       #MyReal	:= 0.0;
       #MyWordsinReal[0]	:= "EPICSToPLC"."Word"[#EPICSToPLCDataBlockOffset + 0];
       #MyWordsinReal[1]	:= "EPICSToPLC"."Word"[#EPICSToPLCDataBlockOffset + 1];
       #"iVolR" := #MyReal;    //EPICSName: iVolR
    Else
       #DEVICE_PARAM_OK := FALSE; //Invalid Hash
    END_IF;
END_FUNCTION_BLOCK
FUNCTION_BLOCK "DEVTYPE_ISRC_LEBT_PS_SOL_STR"
{ S7_Optimized_Access := 'TRUE' }
VERSION : 1.0
   VAR_INPUT
      "CurR-CT" { ExternalAccessible := 'True'; ExternalVisible := 'False'; ExternalWritable := 'False'; } : REAL;   //EPICS Status variable: CurR-CT
      "EnCmdR" { ExternalAccessible := 'True'; ExternalVisible := 'False'; ExternalWritable := 'False'; } : BOOL;   //EPICS Status variable: EnCmdR
      "CurMaxErr" { ExternalAccessible := 'True'; ExternalVisible := 'False'; ExternalWritable := 'False'; } : BOOL;   //EPICS Status variable: CurMaxErr
   EPICSToPLCLength { ExternalAccessible := 'False'; ExternalVisible := 'False'; ExternalWritable := 'False'; } : Int;   // Length of device command register array (in words)
   EPICSToPLCDataBlockOffset { ExternalAccessible := 'False'; ExternalVisible := 'False'; ExternalWritable := 'False'; } : Int;   // Offset in EPICS->PLC comms block where this device data resides (in words)
   EPICSToPLCParametersStart { ExternalAccessible := 'False'; ExternalVisible := 'False'; ExternalWritable := 'False'; } : Int;   // The border offset between the Command and the Parameter area
   PLCToEPICSLength { ExternalAccessible := 'False'; ExternalVisible := 'False'; ExternalWritable := 'False'; } : Int;   // Length of device status register array (in words)
   PLCToEPICSDataBlockOffset { ExternalAccessible := 'False'; ExternalVisible := 'False'; ExternalWritable := 'False'; } : Int;   // Offset in PLC->EPICS comms block where this device data resides (in words)
   END_VAR
   VAR_OUTPUT
      DEVICE_PARAM_OK { ExternalAccessible := 'False'; ExternalVisible := 'False'; ExternalWritable := 'False'; } : Bool;
   END_VAR
   VAR_IN_OUT
   END_VAR
   Var DB_SPECIFIC
      MyWord { ExternalAccessible := 'False'; ExternalVisible := 'False'; ExternalWritable := 'False'; } : Word;
      MyBytesinWord { ExternalAccessible := 'False'; ExternalVisible := 'False'; ExternalWritable := 'False'; } AT MyWord : Array[0..1] of Byte;
      MyBoolsinWord { ExternalAccessible := 'False'; ExternalVisible := 'False'; ExternalWritable := 'False'; } AT MyWord : Array[0..15] of Bool;
      MyDInt { ExternalAccessible := 'False'; ExternalVisible := 'False'; ExternalWritable := 'False'; } : DInt;
      MyWordsinDint { ExternalAccessible := 'False'; ExternalVisible := 'False'; ExternalWritable := 'False'; } AT MyDInt : Array[0..1] of Word;
      MyReal { ExternalAccessible := 'False'; ExternalVisible := 'False'; ExternalWritable := 'False'; } : Real;
      MyWordsinReal { ExternalAccessible := 'False'; ExternalVisible := 'False'; ExternalWritable := 'False'; } AT MyReal : Array[0..1] of Word;
      MyInt { ExternalAccessible := 'False'; ExternalVisible := 'False'; ExternalWritable := 'False'; } : Int;
      MyWordinInt { ExternalAccessible := 'False'; ExternalVisible := 'False'; ExternalWritable := 'False'; } AT MyInt : Word;
      MyDWord { ExternalAccessible := 'False'; ExternalVisible := 'False'; ExternalWritable := 'False'; } : DWord;
      MyWordsinDWord { ExternalAccessible := 'False'; ExternalVisible := 'False'; ExternalWritable := 'False'; } AT MyDWord : Array[0..1] of Word;
      MyTime { ExternalAccessible := 'False'; ExternalVisible := 'False'; ExternalWritable := 'False'; } : Time;
      MyWordsinTime { ExternalAccessible := 'False'; ExternalVisible := 'False'; ExternalWritable := 'False'; } AT MyTime : Array[0..1] of Word;
      MyString { ExternalAccessible := 'False'; ExternalVisible := 'False'; ExternalWritable := 'False'; } : String[40];
      MyWordsinString { ExternalAccessible := 'False'; ExternalVisible := 'False'; ExternalWritable := 'False'; } AT MyString : Array[0..20] of Word;
   END_VAR
   VAR_TEMP
      HashModbus : DInt;
      HashIFA : DInt;
      HashTIAMap : DInt;
      i : Int;
   END_VAR
    //Author: Miklos Boros (miklos.boros@esss.se), Copyrigth 2017-2019 by European Spallation Source, Lund
    //This block was generated by PLCFactory, please don't change it MANUALLY!
    //Input File Name: ISrc-010_Ctrl-PLC-01-template-IFA-20191106135317.ifa
    //Generated: 20191106135317
    //According to HASH: 1347332123
    //Device type: ISRC_LEBT_PS_SOL_STR
    //Description: This function does the variable mapping for a device. All device-variable will be linked to an interface variable defined in this block.

    //********************************************
    //****************HASH check******************
    //********************************************


    #MyWordsinDint[0] := "EPICSToPLC"."Word"[0];
    #MyWordsinDint[1] := "EPICSToPLC"."Word"[1];
    #HashModbus := #MyDInt; //Hash from EPICS/ModbusTCP

    #HashIFA := 1347332123; //Hash from Interface Factory as a constant

    #MyWordsinDint[0] := "PLCToEPICS"."Word"[0];
    #MyWordsinDint[1] := "PLCToEPICS"."Word"[1];
    #HashTIAMap := #MyDInt; //Hash from PLCFactory TIA Map


    IF ((#HashIFA = #HashModbus) AND (#HashModbus = #HashTIAMap)) THEN //Check CRCs
        #DEVICE_PARAM_OK := TRUE;
       //###########################  LEBT Solenoids and Steerers PowerSupply  ##############################
       //###########################
       //STATUS BLOCK
       //###########################

    //********************************************
    //*************STATUS VARIABLES***************
    //********************************************


       #MyReal := #"CurR-CT";    //EPICSName: CurR-CT
       "PLCToEPICS"."Word"[#PLCToEPICSDataBlockOffset + 0] := #MyWordsinReal[0];
       "PLCToEPICS"."Word"[#PLCToEPICSDataBlockOffset + 1] := #MyWordsinReal[1];

       #MyWord := W#0;
       #MyBoolsinWord[8] := #"EnCmdR";    //EPICSName: EnCmdR
       #MyBoolsinWord[9] := #"CurMaxErr";    //EPICSName: CurMaxErr
       "PLCToEPICS"."Word"[#PLCToEPICSDataBlockOffset + 2] := #MyWord;
    Else
       #DEVICE_PARAM_OK := FALSE; //Invalid Hash
    END_IF;
END_FUNCTION_BLOCK
FUNCTION_BLOCK "DEVTYPE_ISRC_LEBT_PlasCh"
{ S7_Optimized_Access := 'TRUE' }
VERSION : 1.0
   VAR_INPUT
      "WtrFlowOK" { ExternalAccessible := 'True'; ExternalVisible := 'False'; ExternalWritable := 'False'; } : BOOL;   //EPICS Status variable: WtrFlowOK
   EPICSToPLCLength { ExternalAccessible := 'False'; ExternalVisible := 'False'; ExternalWritable := 'False'; } : Int;   // Length of device command register array (in words)
   EPICSToPLCDataBlockOffset { ExternalAccessible := 'False'; ExternalVisible := 'False'; ExternalWritable := 'False'; } : Int;   // Offset in EPICS->PLC comms block where this device data resides (in words)
   EPICSToPLCParametersStart { ExternalAccessible := 'False'; ExternalVisible := 'False'; ExternalWritable := 'False'; } : Int;   // The border offset between the Command and the Parameter area
   PLCToEPICSLength { ExternalAccessible := 'False'; ExternalVisible := 'False'; ExternalWritable := 'False'; } : Int;   // Length of device status register array (in words)
   PLCToEPICSDataBlockOffset { ExternalAccessible := 'False'; ExternalVisible := 'False'; ExternalWritable := 'False'; } : Int;   // Offset in PLC->EPICS comms block where this device data resides (in words)
   END_VAR
   VAR_OUTPUT
      DEVICE_PARAM_OK { ExternalAccessible := 'False'; ExternalVisible := 'False'; ExternalWritable := 'False'; } : Bool;
   END_VAR
   VAR_IN_OUT
   END_VAR
   Var DB_SPECIFIC
      MyWord { ExternalAccessible := 'False'; ExternalVisible := 'False'; ExternalWritable := 'False'; } : Word;
      MyBytesinWord { ExternalAccessible := 'False'; ExternalVisible := 'False'; ExternalWritable := 'False'; } AT MyWord : Array[0..1] of Byte;
      MyBoolsinWord { ExternalAccessible := 'False'; ExternalVisible := 'False'; ExternalWritable := 'False'; } AT MyWord : Array[0..15] of Bool;
      MyDInt { ExternalAccessible := 'False'; ExternalVisible := 'False'; ExternalWritable := 'False'; } : DInt;
      MyWordsinDint { ExternalAccessible := 'False'; ExternalVisible := 'False'; ExternalWritable := 'False'; } AT MyDInt : Array[0..1] of Word;
      MyReal { ExternalAccessible := 'False'; ExternalVisible := 'False'; ExternalWritable := 'False'; } : Real;
      MyWordsinReal { ExternalAccessible := 'False'; ExternalVisible := 'False'; ExternalWritable := 'False'; } AT MyReal : Array[0..1] of Word;
      MyInt { ExternalAccessible := 'False'; ExternalVisible := 'False'; ExternalWritable := 'False'; } : Int;
      MyWordinInt { ExternalAccessible := 'False'; ExternalVisible := 'False'; ExternalWritable := 'False'; } AT MyInt : Word;
      MyDWord { ExternalAccessible := 'False'; ExternalVisible := 'False'; ExternalWritable := 'False'; } : DWord;
      MyWordsinDWord { ExternalAccessible := 'False'; ExternalVisible := 'False'; ExternalWritable := 'False'; } AT MyDWord : Array[0..1] of Word;
      MyTime { ExternalAccessible := 'False'; ExternalVisible := 'False'; ExternalWritable := 'False'; } : Time;
      MyWordsinTime { ExternalAccessible := 'False'; ExternalVisible := 'False'; ExternalWritable := 'False'; } AT MyTime : Array[0..1] of Word;
      MyString { ExternalAccessible := 'False'; ExternalVisible := 'False'; ExternalWritable := 'False'; } : String[40];
      MyWordsinString { ExternalAccessible := 'False'; ExternalVisible := 'False'; ExternalWritable := 'False'; } AT MyString : Array[0..20] of Word;
   END_VAR
   VAR_TEMP
      HashModbus : DInt;
      HashIFA : DInt;
      HashTIAMap : DInt;
      i : Int;
   END_VAR
    //Author: Miklos Boros (miklos.boros@esss.se), Copyrigth 2017-2019 by European Spallation Source, Lund
    //This block was generated by PLCFactory, please don't change it MANUALLY!
    //Input File Name: ISrc-010_Ctrl-PLC-01-template-IFA-20191106135317.ifa
    //Generated: 20191106135317
    //According to HASH: 1347332123
    //Device type: ISRC_LEBT_PlasCh
    //Description: This function does the variable mapping for a device. All device-variable will be linked to an interface variable defined in this block.

    //********************************************
    //****************HASH check******************
    //********************************************


    #MyWordsinDint[0] := "EPICSToPLC"."Word"[0];
    #MyWordsinDint[1] := "EPICSToPLC"."Word"[1];
    #HashModbus := #MyDInt; //Hash from EPICS/ModbusTCP

    #HashIFA := 1347332123; //Hash from Interface Factory as a constant

    #MyWordsinDint[0] := "PLCToEPICS"."Word"[0];
    #MyWordsinDint[1] := "PLCToEPICS"."Word"[1];
    #HashTIAMap := #MyDInt; //Hash from PLCFactory TIA Map


    IF ((#HashIFA = #HashModbus) AND (#HashModbus = #HashTIAMap)) THEN //Check CRCs
        #DEVICE_PARAM_OK := TRUE;
       //###########################  ISRC Plasma Chamber  ##############################
       //###########################
       //STATUS BLOCK
       //###########################

    //********************************************
    //*************STATUS VARIABLES***************
    //********************************************


       #MyWord := W#0;
       #MyBoolsinWord[8] := #"WtrFlowOK";    //EPICSName: WtrFlowOK
       "PLCToEPICS"."Word"[#PLCToEPICSDataBlockOffset + 0] := #MyWord;
    Else
       #DEVICE_PARAM_OK := FALSE; //Invalid Hash
    END_IF;
END_FUNCTION_BLOCK
FUNCTION_BLOCK "DEVTYPE_ISRC_LEBT_REP"
{ S7_Optimized_Access := 'TRUE' }
VERSION : 1.0
   VAR_INPUT
      "WtrFlowOK" { ExternalAccessible := 'True'; ExternalVisible := 'False'; ExternalWritable := 'False'; } : BOOL;   //EPICS Status variable: WtrFlowOK
   EPICSToPLCLength { ExternalAccessible := 'False'; ExternalVisible := 'False'; ExternalWritable := 'False'; } : Int;   // Length of device command register array (in words)
   EPICSToPLCDataBlockOffset { ExternalAccessible := 'False'; ExternalVisible := 'False'; ExternalWritable := 'False'; } : Int;   // Offset in EPICS->PLC comms block where this device data resides (in words)
   EPICSToPLCParametersStart { ExternalAccessible := 'False'; ExternalVisible := 'False'; ExternalWritable := 'False'; } : Int;   // The border offset between the Command and the Parameter area
   PLCToEPICSLength { ExternalAccessible := 'False'; ExternalVisible := 'False'; ExternalWritable := 'False'; } : Int;   // Length of device status register array (in words)
   PLCToEPICSDataBlockOffset { ExternalAccessible := 'False'; ExternalVisible := 'False'; ExternalWritable := 'False'; } : Int;   // Offset in PLC->EPICS comms block where this device data resides (in words)
   END_VAR
   VAR_OUTPUT
      DEVICE_PARAM_OK { ExternalAccessible := 'False'; ExternalVisible := 'False'; ExternalWritable := 'False'; } : Bool;
   END_VAR
   VAR_IN_OUT
   END_VAR
   Var DB_SPECIFIC
      MyWord { ExternalAccessible := 'False'; ExternalVisible := 'False'; ExternalWritable := 'False'; } : Word;
      MyBytesinWord { ExternalAccessible := 'False'; ExternalVisible := 'False'; ExternalWritable := 'False'; } AT MyWord : Array[0..1] of Byte;
      MyBoolsinWord { ExternalAccessible := 'False'; ExternalVisible := 'False'; ExternalWritable := 'False'; } AT MyWord : Array[0..15] of Bool;
      MyDInt { ExternalAccessible := 'False'; ExternalVisible := 'False'; ExternalWritable := 'False'; } : DInt;
      MyWordsinDint { ExternalAccessible := 'False'; ExternalVisible := 'False'; ExternalWritable := 'False'; } AT MyDInt : Array[0..1] of Word;
      MyReal { ExternalAccessible := 'False'; ExternalVisible := 'False'; ExternalWritable := 'False'; } : Real;
      MyWordsinReal { ExternalAccessible := 'False'; ExternalVisible := 'False'; ExternalWritable := 'False'; } AT MyReal : Array[0..1] of Word;
      MyInt { ExternalAccessible := 'False'; ExternalVisible := 'False'; ExternalWritable := 'False'; } : Int;
      MyWordinInt { ExternalAccessible := 'False'; ExternalVisible := 'False'; ExternalWritable := 'False'; } AT MyInt : Word;
      MyDWord { ExternalAccessible := 'False'; ExternalVisible := 'False'; ExternalWritable := 'False'; } : DWord;
      MyWordsinDWord { ExternalAccessible := 'False'; ExternalVisible := 'False'; ExternalWritable := 'False'; } AT MyDWord : Array[0..1] of Word;
      MyTime { ExternalAccessible := 'False'; ExternalVisible := 'False'; ExternalWritable := 'False'; } : Time;
      MyWordsinTime { ExternalAccessible := 'False'; ExternalVisible := 'False'; ExternalWritable := 'False'; } AT MyTime : Array[0..1] of Word;
      MyString { ExternalAccessible := 'False'; ExternalVisible := 'False'; ExternalWritable := 'False'; } : String[40];
      MyWordsinString { ExternalAccessible := 'False'; ExternalVisible := 'False'; ExternalWritable := 'False'; } AT MyString : Array[0..20] of Word;
   END_VAR
   VAR_TEMP
      HashModbus : DInt;
      HashIFA : DInt;
      HashTIAMap : DInt;
      i : Int;
   END_VAR
    //Author: Miklos Boros (miklos.boros@esss.se), Copyrigth 2017-2019 by European Spallation Source, Lund
    //This block was generated by PLCFactory, please don't change it MANUALLY!
    //Input File Name: ISrc-010_Ctrl-PLC-01-template-IFA-20191106135317.ifa
    //Generated: 20191106135317
    //According to HASH: 1347332123
    //Device type: ISRC_LEBT_REP
    //Description: This function does the variable mapping for a device. All device-variable will be linked to an interface variable defined in this block.

    //********************************************
    //****************HASH check******************
    //********************************************


    #MyWordsinDint[0] := "EPICSToPLC"."Word"[0];
    #MyWordsinDint[1] := "EPICSToPLC"."Word"[1];
    #HashModbus := #MyDInt; //Hash from EPICS/ModbusTCP

    #HashIFA := 1347332123; //Hash from Interface Factory as a constant

    #MyWordsinDint[0] := "PLCToEPICS"."Word"[0];
    #MyWordsinDint[1] := "PLCToEPICS"."Word"[1];
    #HashTIAMap := #MyDInt; //Hash from PLCFactory TIA Map


    IF ((#HashIFA = #HashModbus) AND (#HashModbus = #HashTIAMap)) THEN //Check CRCs
        #DEVICE_PARAM_OK := TRUE;
       //###########################  ISrc and LEBT Repeller  ##############################
       //###########################
       //STATUS BLOCK
       //###########################

    //********************************************
    //*************STATUS VARIABLES***************
    //********************************************


       #MyWord := W#0;
       #MyBoolsinWord[8] := #"WtrFlowOK";    //EPICSName: WtrFlowOK
       "PLCToEPICS"."Word"[#PLCToEPICSDataBlockOffset + 0] := #MyWord;
    Else
       #DEVICE_PARAM_OK := FALSE; //Invalid Hash
    END_IF;
END_FUNCTION_BLOCK
FUNCTION_BLOCK "DEVTYPE_ISRC_LEBT_STR"
{ S7_Optimized_Access := 'TRUE' }
VERSION : 1.0
   VAR_INPUT
      "PolR" { ExternalAccessible := 'True'; ExternalVisible := 'False'; ExternalWritable := 'False'; } : BOOL;   //EPICS Status variable: PolR
   EPICSToPLCLength { ExternalAccessible := 'False'; ExternalVisible := 'False'; ExternalWritable := 'False'; } : Int;   // Length of device command register array (in words)
   EPICSToPLCDataBlockOffset { ExternalAccessible := 'False'; ExternalVisible := 'False'; ExternalWritable := 'False'; } : Int;   // Offset in EPICS->PLC comms block where this device data resides (in words)
   EPICSToPLCParametersStart { ExternalAccessible := 'False'; ExternalVisible := 'False'; ExternalWritable := 'False'; } : Int;   // The border offset between the Command and the Parameter area
   PLCToEPICSLength { ExternalAccessible := 'False'; ExternalVisible := 'False'; ExternalWritable := 'False'; } : Int;   // Length of device status register array (in words)
   PLCToEPICSDataBlockOffset { ExternalAccessible := 'False'; ExternalVisible := 'False'; ExternalWritable := 'False'; } : Int;   // Offset in PLC->EPICS comms block where this device data resides (in words)
   END_VAR
   VAR_OUTPUT
      "PolPosCmd" { ExternalAccessible := 'True'; ExternalVisible := 'False'; ExternalWritable := 'False'; } : BOOL;   //EPICS Command variable: PolPosCmd
      "PolNegCmd" { ExternalAccessible := 'True'; ExternalVisible := 'False'; ExternalWritable := 'False'; } : BOOL;   //EPICS Command variable: PolNegCmd
      DEVICE_PARAM_OK { ExternalAccessible := 'False'; ExternalVisible := 'False'; ExternalWritable := 'False'; } : Bool;
   END_VAR
   VAR_IN_OUT
   END_VAR
   Var DB_SPECIFIC
      MyWord { ExternalAccessible := 'False'; ExternalVisible := 'False'; ExternalWritable := 'False'; } : Word;
      MyBytesinWord { ExternalAccessible := 'False'; ExternalVisible := 'False'; ExternalWritable := 'False'; } AT MyWord : Array[0..1] of Byte;
      MyBoolsinWord { ExternalAccessible := 'False'; ExternalVisible := 'False'; ExternalWritable := 'False'; } AT MyWord : Array[0..15] of Bool;
      MyDInt { ExternalAccessible := 'False'; ExternalVisible := 'False'; ExternalWritable := 'False'; } : DInt;
      MyWordsinDint { ExternalAccessible := 'False'; ExternalVisible := 'False'; ExternalWritable := 'False'; } AT MyDInt : Array[0..1] of Word;
      MyReal { ExternalAccessible := 'False'; ExternalVisible := 'False'; ExternalWritable := 'False'; } : Real;
      MyWordsinReal { ExternalAccessible := 'False'; ExternalVisible := 'False'; ExternalWritable := 'False'; } AT MyReal : Array[0..1] of Word;
      MyInt { ExternalAccessible := 'False'; ExternalVisible := 'False'; ExternalWritable := 'False'; } : Int;
      MyWordinInt { ExternalAccessible := 'False'; ExternalVisible := 'False'; ExternalWritable := 'False'; } AT MyInt : Word;
      MyDWord { ExternalAccessible := 'False'; ExternalVisible := 'False'; ExternalWritable := 'False'; } : DWord;
      MyWordsinDWord { ExternalAccessible := 'False'; ExternalVisible := 'False'; ExternalWritable := 'False'; } AT MyDWord : Array[0..1] of Word;
      MyTime { ExternalAccessible := 'False'; ExternalVisible := 'False'; ExternalWritable := 'False'; } : Time;
      MyWordsinTime { ExternalAccessible := 'False'; ExternalVisible := 'False'; ExternalWritable := 'False'; } AT MyTime : Array[0..1] of Word;
      MyString { ExternalAccessible := 'False'; ExternalVisible := 'False'; ExternalWritable := 'False'; } : String[40];
      MyWordsinString { ExternalAccessible := 'False'; ExternalVisible := 'False'; ExternalWritable := 'False'; } AT MyString : Array[0..20] of Word;
   END_VAR
   VAR_TEMP
      HashModbus : DInt;
      HashIFA : DInt;
      HashTIAMap : DInt;
      i : Int;
   END_VAR
    //Author: Miklos Boros (miklos.boros@esss.se), Copyrigth 2017-2019 by European Spallation Source, Lund
    //This block was generated by PLCFactory, please don't change it MANUALLY!
    //Input File Name: ISrc-010_Ctrl-PLC-01-template-IFA-20191106135317.ifa
    //Generated: 20191106135317
    //According to HASH: 1347332123
    //Device type: ISRC_LEBT_STR
    //Description: This function does the variable mapping for a device. All device-variable will be linked to an interface variable defined in this block.

    //********************************************
    //****************HASH check******************
    //********************************************


    #MyWordsinDint[0] := "EPICSToPLC"."Word"[0];
    #MyWordsinDint[1] := "EPICSToPLC"."Word"[1];
    #HashModbus := #MyDInt; //Hash from EPICS/ModbusTCP

    #HashIFA := 1347332123; //Hash from Interface Factory as a constant

    #MyWordsinDint[0] := "PLCToEPICS"."Word"[0];
    #MyWordsinDint[1] := "PLCToEPICS"."Word"[1];
    #HashTIAMap := #MyDInt; //Hash from PLCFactory TIA Map


    IF ((#HashIFA = #HashModbus) AND (#HashModbus = #HashTIAMap)) THEN //Check CRCs
        #DEVICE_PARAM_OK := TRUE;
       //#############################  LEBT Steerer  ##############################
       //###########################
       //STATUS BLOCK
       //###########################

    //********************************************
    //*************STATUS VARIABLES***************
    //********************************************


       #MyWord := W#0;
       #MyBoolsinWord[8] := #"PolR";    //EPICSName: PolR
       "PLCToEPICS"."Word"[#PLCToEPICSDataBlockOffset + 0] := #MyWord;

    //********************************************
    //*************COMMAND VARIABLES**************
    //********************************************


       #MyWord := "EPICSToPLC"."Word"[#EPICSToPLCDataBlockOffset + 0];
       IF (NOT "Utilities".TestInProgress) THEN
       	"EPICSToPLC"."Word"[#EPICSToPLCDataBlockOffset + 0] := 0;
       END_IF;
       #"PolPosCmd" := #MyBoolsinWord[8];    //EPICSName: PolPosCmd
       #"PolNegCmd" := #MyBoolsinWord[9];    //EPICSName: PolNegCmd
    Else
       #DEVICE_PARAM_OK := FALSE; //Invalid Hash
    END_IF;
END_FUNCTION_BLOCK
FUNCTION_BLOCK "DEVTYPE_ISRC_LEBT_VAC_VVA"
{ S7_Optimized_Access := 'TRUE' }
VERSION : 1.0
   VAR_INPUT
      "OpenR" { ExternalAccessible := 'True'; ExternalVisible := 'False'; ExternalWritable := 'False'; } : BOOL;   //EPICS Status variable: OpenR
      "OpenCmdRB" { ExternalAccessible := 'True'; ExternalVisible := 'False'; ExternalWritable := 'False'; } : BOOL;   //EPICS Status variable: OpenCmdRB
   EPICSToPLCLength { ExternalAccessible := 'False'; ExternalVisible := 'False'; ExternalWritable := 'False'; } : Int;   // Length of device command register array (in words)
   EPICSToPLCDataBlockOffset { ExternalAccessible := 'False'; ExternalVisible := 'False'; ExternalWritable := 'False'; } : Int;   // Offset in EPICS->PLC comms block where this device data resides (in words)
   EPICSToPLCParametersStart { ExternalAccessible := 'False'; ExternalVisible := 'False'; ExternalWritable := 'False'; } : Int;   // The border offset between the Command and the Parameter area
   PLCToEPICSLength { ExternalAccessible := 'False'; ExternalVisible := 'False'; ExternalWritable := 'False'; } : Int;   // Length of device status register array (in words)
   PLCToEPICSDataBlockOffset { ExternalAccessible := 'False'; ExternalVisible := 'False'; ExternalWritable := 'False'; } : Int;   // Offset in PLC->EPICS comms block where this device data resides (in words)
   END_VAR
   VAR_OUTPUT
      "OpenCmd" { ExternalAccessible := 'True'; ExternalVisible := 'False'; ExternalWritable := 'False'; } : BOOL;   //EPICS Command variable: OpenCmd
      "CloseCmd" { ExternalAccessible := 'True'; ExternalVisible := 'False'; ExternalWritable := 'False'; } : BOOL;   //EPICS Command variable: CloseCmd
      DEVICE_PARAM_OK { ExternalAccessible := 'False'; ExternalVisible := 'False'; ExternalWritable := 'False'; } : Bool;
   END_VAR
   VAR_IN_OUT
   END_VAR
   Var DB_SPECIFIC
      MyWord { ExternalAccessible := 'False'; ExternalVisible := 'False'; ExternalWritable := 'False'; } : Word;
      MyBytesinWord { ExternalAccessible := 'False'; ExternalVisible := 'False'; ExternalWritable := 'False'; } AT MyWord : Array[0..1] of Byte;
      MyBoolsinWord { ExternalAccessible := 'False'; ExternalVisible := 'False'; ExternalWritable := 'False'; } AT MyWord : Array[0..15] of Bool;
      MyDInt { ExternalAccessible := 'False'; ExternalVisible := 'False'; ExternalWritable := 'False'; } : DInt;
      MyWordsinDint { ExternalAccessible := 'False'; ExternalVisible := 'False'; ExternalWritable := 'False'; } AT MyDInt : Array[0..1] of Word;
      MyReal { ExternalAccessible := 'False'; ExternalVisible := 'False'; ExternalWritable := 'False'; } : Real;
      MyWordsinReal { ExternalAccessible := 'False'; ExternalVisible := 'False'; ExternalWritable := 'False'; } AT MyReal : Array[0..1] of Word;
      MyInt { ExternalAccessible := 'False'; ExternalVisible := 'False'; ExternalWritable := 'False'; } : Int;
      MyWordinInt { ExternalAccessible := 'False'; ExternalVisible := 'False'; ExternalWritable := 'False'; } AT MyInt : Word;
      MyDWord { ExternalAccessible := 'False'; ExternalVisible := 'False'; ExternalWritable := 'False'; } : DWord;
      MyWordsinDWord { ExternalAccessible := 'False'; ExternalVisible := 'False'; ExternalWritable := 'False'; } AT MyDWord : Array[0..1] of Word;
      MyTime { ExternalAccessible := 'False'; ExternalVisible := 'False'; ExternalWritable := 'False'; } : Time;
      MyWordsinTime { ExternalAccessible := 'False'; ExternalVisible := 'False'; ExternalWritable := 'False'; } AT MyTime : Array[0..1] of Word;
      MyString { ExternalAccessible := 'False'; ExternalVisible := 'False'; ExternalWritable := 'False'; } : String[40];
      MyWordsinString { ExternalAccessible := 'False'; ExternalVisible := 'False'; ExternalWritable := 'False'; } AT MyString : Array[0..20] of Word;
   END_VAR
   VAR_TEMP
      HashModbus : DInt;
      HashIFA : DInt;
      HashTIAMap : DInt;
      i : Int;
   END_VAR
    //Author: Miklos Boros (miklos.boros@esss.se), Copyrigth 2017-2019 by European Spallation Source, Lund
    //This block was generated by PLCFactory, please don't change it MANUALLY!
    //Input File Name: ISrc-010_Ctrl-PLC-01-template-IFA-20191106135317.ifa
    //Generated: 20191106135317
    //According to HASH: 1347332123
    //Device type: ISRC_LEBT_VAC_VVA
    //Description: This function does the variable mapping for a device. All device-variable will be linked to an interface variable defined in this block.

    //********************************************
    //****************HASH check******************
    //********************************************


    #MyWordsinDint[0] := "EPICSToPLC"."Word"[0];
    #MyWordsinDint[1] := "EPICSToPLC"."Word"[1];
    #HashModbus := #MyDInt; //Hash from EPICS/ModbusTCP

    #HashIFA := 1347332123; //Hash from Interface Factory as a constant

    #MyWordsinDint[0] := "PLCToEPICS"."Word"[0];
    #MyWordsinDint[1] := "PLCToEPICS"."Word"[1];
    #HashTIAMap := #MyDInt; //Hash from PLCFactory TIA Map


    IF ((#HashIFA = #HashModbus) AND (#HashModbus = #HashTIAMap)) THEN //Check CRCs
        #DEVICE_PARAM_OK := TRUE;
       //###########################  ISRC_LEBT H2 valve in HV platform  ##############################
       //###########################
       //STATUS BLOCK
       //###########################

    //********************************************
    //*************STATUS VARIABLES***************
    //********************************************


       #MyWord := W#0;
       #MyBoolsinWord[8] := #"OpenR";    //EPICSName: OpenR
       #MyBoolsinWord[9] := #"OpenCmdRB";    //EPICSName: OpenCmdRB
       "PLCToEPICS"."Word"[#PLCToEPICSDataBlockOffset + 0] := #MyWord;

    //********************************************
    //*************COMMAND VARIABLES**************
    //********************************************


       #MyWord := "EPICSToPLC"."Word"[#EPICSToPLCDataBlockOffset + 0];
       IF (NOT "Utilities".TestInProgress) THEN
       	"EPICSToPLC"."Word"[#EPICSToPLCDataBlockOffset + 0] := 0;
       END_IF;
       #"OpenCmd" := #MyBoolsinWord[8];    //EPICSName: OpenCmd
       #"CloseCmd" := #MyBoolsinWord[9];    //EPICSName: CloseCmd
    Else
       #DEVICE_PARAM_OK := FALSE; //Invalid Hash
    END_IF;
END_FUNCTION_BLOCK
FUNCTION_BLOCK "DEVTYPE_ISRC_LEBT_WTRC_PRES"
{ S7_Optimized_Access := 'TRUE' }
VERSION : 1.0
   VAR_INPUT
      "PresR" { ExternalAccessible := 'True'; ExternalVisible := 'False'; ExternalWritable := 'False'; } : REAL;   //EPICS Status variable: PresR
   EPICSToPLCLength { ExternalAccessible := 'False'; ExternalVisible := 'False'; ExternalWritable := 'False'; } : Int;   // Length of device command register array (in words)
   EPICSToPLCDataBlockOffset { ExternalAccessible := 'False'; ExternalVisible := 'False'; ExternalWritable := 'False'; } : Int;   // Offset in EPICS->PLC comms block where this device data resides (in words)
   EPICSToPLCParametersStart { ExternalAccessible := 'False'; ExternalVisible := 'False'; ExternalWritable := 'False'; } : Int;   // The border offset between the Command and the Parameter area
   PLCToEPICSLength { ExternalAccessible := 'False'; ExternalVisible := 'False'; ExternalWritable := 'False'; } : Int;   // Length of device status register array (in words)
   PLCToEPICSDataBlockOffset { ExternalAccessible := 'False'; ExternalVisible := 'False'; ExternalWritable := 'False'; } : Int;   // Offset in PLC->EPICS comms block where this device data resides (in words)
   END_VAR
   VAR_OUTPUT
      DEVICE_PARAM_OK { ExternalAccessible := 'False'; ExternalVisible := 'False'; ExternalWritable := 'False'; } : Bool;
   END_VAR
   VAR_IN_OUT
   END_VAR
   Var DB_SPECIFIC
      MyWord { ExternalAccessible := 'False'; ExternalVisible := 'False'; ExternalWritable := 'False'; } : Word;
      MyBytesinWord { ExternalAccessible := 'False'; ExternalVisible := 'False'; ExternalWritable := 'False'; } AT MyWord : Array[0..1] of Byte;
      MyBoolsinWord { ExternalAccessible := 'False'; ExternalVisible := 'False'; ExternalWritable := 'False'; } AT MyWord : Array[0..15] of Bool;
      MyDInt { ExternalAccessible := 'False'; ExternalVisible := 'False'; ExternalWritable := 'False'; } : DInt;
      MyWordsinDint { ExternalAccessible := 'False'; ExternalVisible := 'False'; ExternalWritable := 'False'; } AT MyDInt : Array[0..1] of Word;
      MyReal { ExternalAccessible := 'False'; ExternalVisible := 'False'; ExternalWritable := 'False'; } : Real;
      MyWordsinReal { ExternalAccessible := 'False'; ExternalVisible := 'False'; ExternalWritable := 'False'; } AT MyReal : Array[0..1] of Word;
      MyInt { ExternalAccessible := 'False'; ExternalVisible := 'False'; ExternalWritable := 'False'; } : Int;
      MyWordinInt { ExternalAccessible := 'False'; ExternalVisible := 'False'; ExternalWritable := 'False'; } AT MyInt : Word;
      MyDWord { ExternalAccessible := 'False'; ExternalVisible := 'False'; ExternalWritable := 'False'; } : DWord;
      MyWordsinDWord { ExternalAccessible := 'False'; ExternalVisible := 'False'; ExternalWritable := 'False'; } AT MyDWord : Array[0..1] of Word;
      MyTime { ExternalAccessible := 'False'; ExternalVisible := 'False'; ExternalWritable := 'False'; } : Time;
      MyWordsinTime { ExternalAccessible := 'False'; ExternalVisible := 'False'; ExternalWritable := 'False'; } AT MyTime : Array[0..1] of Word;
      MyString { ExternalAccessible := 'False'; ExternalVisible := 'False'; ExternalWritable := 'False'; } : String[40];
      MyWordsinString { ExternalAccessible := 'False'; ExternalVisible := 'False'; ExternalWritable := 'False'; } AT MyString : Array[0..20] of Word;
   END_VAR
   VAR_TEMP
      HashModbus : DInt;
      HashIFA : DInt;
      HashTIAMap : DInt;
      i : Int;
   END_VAR
    //Author: Miklos Boros (miklos.boros@esss.se), Copyrigth 2017-2019 by European Spallation Source, Lund
    //This block was generated by PLCFactory, please don't change it MANUALLY!
    //Input File Name: ISrc-010_Ctrl-PLC-01-template-IFA-20191106135317.ifa
    //Generated: 20191106135317
    //According to HASH: 1347332123
    //Device type: ISRC_LEBT_WTRC_PRES
    //Description: This function does the variable mapping for a device. All device-variable will be linked to an interface variable defined in this block.

    //********************************************
    //****************HASH check******************
    //********************************************


    #MyWordsinDint[0] := "EPICSToPLC"."Word"[0];
    #MyWordsinDint[1] := "EPICSToPLC"."Word"[1];
    #HashModbus := #MyDInt; //Hash from EPICS/ModbusTCP

    #HashIFA := 1347332123; //Hash from Interface Factory as a constant

    #MyWordsinDint[0] := "PLCToEPICS"."Word"[0];
    #MyWordsinDint[1] := "PLCToEPICS"."Word"[1];
    #HashTIAMap := #MyDInt; //Hash from PLCFactory TIA Map


    IF ((#HashIFA = #HashModbus) AND (#HashModbus = #HashTIAMap)) THEN //Check CRCs
        #DEVICE_PARAM_OK := TRUE;
       //###########################  ISRC_LEBT Water Cooling Pressure Transmitter  ##############################
       //###########################
       //STATUS BLOCK
       //###########################

    //********************************************
    //*************STATUS VARIABLES***************
    //********************************************


       #MyReal := #"PresR";    //EPICSName: PresR
       "PLCToEPICS"."Word"[#PLCToEPICSDataBlockOffset + 0] := #MyWordsinReal[0];
       "PLCToEPICS"."Word"[#PLCToEPICSDataBlockOffset + 1] := #MyWordsinReal[1];
    Else
       #DEVICE_PARAM_OK := FALSE; //Invalid Hash
    END_IF;
END_FUNCTION_BLOCK
FUNCTION_BLOCK "DEVTYPE_ISRC_LEBT_WTRC_TEMP"
{ S7_Optimized_Access := 'TRUE' }
VERSION : 1.0
   VAR_INPUT
      "TempR" { ExternalAccessible := 'True'; ExternalVisible := 'False'; ExternalWritable := 'False'; } : REAL;   //EPICS Status variable: TempR
      "WtrTempMaxErr" { ExternalAccessible := 'True'; ExternalVisible := 'False'; ExternalWritable := 'False'; } : BOOL;   //EPICS Status variable: WtrTempMaxErr
   EPICSToPLCLength { ExternalAccessible := 'False'; ExternalVisible := 'False'; ExternalWritable := 'False'; } : Int;   // Length of device command register array (in words)
   EPICSToPLCDataBlockOffset { ExternalAccessible := 'False'; ExternalVisible := 'False'; ExternalWritable := 'False'; } : Int;   // Offset in EPICS->PLC comms block where this device data resides (in words)
   EPICSToPLCParametersStart { ExternalAccessible := 'False'; ExternalVisible := 'False'; ExternalWritable := 'False'; } : Int;   // The border offset between the Command and the Parameter area
   PLCToEPICSLength { ExternalAccessible := 'False'; ExternalVisible := 'False'; ExternalWritable := 'False'; } : Int;   // Length of device status register array (in words)
   PLCToEPICSDataBlockOffset { ExternalAccessible := 'False'; ExternalVisible := 'False'; ExternalWritable := 'False'; } : Int;   // Offset in PLC->EPICS comms block where this device data resides (in words)
   END_VAR
   VAR_OUTPUT
      DEVICE_PARAM_OK { ExternalAccessible := 'False'; ExternalVisible := 'False'; ExternalWritable := 'False'; } : Bool;
   END_VAR
   VAR_IN_OUT
   END_VAR
   Var DB_SPECIFIC
      MyWord { ExternalAccessible := 'False'; ExternalVisible := 'False'; ExternalWritable := 'False'; } : Word;
      MyBytesinWord { ExternalAccessible := 'False'; ExternalVisible := 'False'; ExternalWritable := 'False'; } AT MyWord : Array[0..1] of Byte;
      MyBoolsinWord { ExternalAccessible := 'False'; ExternalVisible := 'False'; ExternalWritable := 'False'; } AT MyWord : Array[0..15] of Bool;
      MyDInt { ExternalAccessible := 'False'; ExternalVisible := 'False'; ExternalWritable := 'False'; } : DInt;
      MyWordsinDint { ExternalAccessible := 'False'; ExternalVisible := 'False'; ExternalWritable := 'False'; } AT MyDInt : Array[0..1] of Word;
      MyReal { ExternalAccessible := 'False'; ExternalVisible := 'False'; ExternalWritable := 'False'; } : Real;
      MyWordsinReal { ExternalAccessible := 'False'; ExternalVisible := 'False'; ExternalWritable := 'False'; } AT MyReal : Array[0..1] of Word;
      MyInt { ExternalAccessible := 'False'; ExternalVisible := 'False'; ExternalWritable := 'False'; } : Int;
      MyWordinInt { ExternalAccessible := 'False'; ExternalVisible := 'False'; ExternalWritable := 'False'; } AT MyInt : Word;
      MyDWord { ExternalAccessible := 'False'; ExternalVisible := 'False'; ExternalWritable := 'False'; } : DWord;
      MyWordsinDWord { ExternalAccessible := 'False'; ExternalVisible := 'False'; ExternalWritable := 'False'; } AT MyDWord : Array[0..1] of Word;
      MyTime { ExternalAccessible := 'False'; ExternalVisible := 'False'; ExternalWritable := 'False'; } : Time;
      MyWordsinTime { ExternalAccessible := 'False'; ExternalVisible := 'False'; ExternalWritable := 'False'; } AT MyTime : Array[0..1] of Word;
      MyString { ExternalAccessible := 'False'; ExternalVisible := 'False'; ExternalWritable := 'False'; } : String[40];
      MyWordsinString { ExternalAccessible := 'False'; ExternalVisible := 'False'; ExternalWritable := 'False'; } AT MyString : Array[0..20] of Word;
   END_VAR
   VAR_TEMP
      HashModbus : DInt;
      HashIFA : DInt;
      HashTIAMap : DInt;
      i : Int;
   END_VAR
    //Author: Miklos Boros (miklos.boros@esss.se), Copyrigth 2017-2019 by European Spallation Source, Lund
    //This block was generated by PLCFactory, please don't change it MANUALLY!
    //Input File Name: ISrc-010_Ctrl-PLC-01-template-IFA-20191106135317.ifa
    //Generated: 20191106135317
    //According to HASH: 1347332123
    //Device type: ISRC_LEBT_WTRC_TEMP
    //Description: This function does the variable mapping for a device. All device-variable will be linked to an interface variable defined in this block.

    //********************************************
    //****************HASH check******************
    //********************************************


    #MyWordsinDint[0] := "EPICSToPLC"."Word"[0];
    #MyWordsinDint[1] := "EPICSToPLC"."Word"[1];
    #HashModbus := #MyDInt; //Hash from EPICS/ModbusTCP

    #HashIFA := 1347332123; //Hash from Interface Factory as a constant

    #MyWordsinDint[0] := "PLCToEPICS"."Word"[0];
    #MyWordsinDint[1] := "PLCToEPICS"."Word"[1];
    #HashTIAMap := #MyDInt; //Hash from PLCFactory TIA Map


    IF ((#HashIFA = #HashModbus) AND (#HashModbus = #HashTIAMap)) THEN //Check CRCs
        #DEVICE_PARAM_OK := TRUE;
       //###########################  ISRC_LEBT Water Cooling Temperature Transmitter  ##############################
       //###########################
       //STATUS BLOCK
       //###########################

    //********************************************
    //*************STATUS VARIABLES***************
    //********************************************


       #MyReal := #"TempR";    //EPICSName: TempR
       "PLCToEPICS"."Word"[#PLCToEPICSDataBlockOffset + 0] := #MyWordsinReal[0];
       "PLCToEPICS"."Word"[#PLCToEPICSDataBlockOffset + 1] := #MyWordsinReal[1];

       #MyWord := W#0;
       #MyBoolsinWord[8] := #"WtrTempMaxErr";    //EPICSName: WtrTempMaxErr
       "PLCToEPICS"."Word"[#PLCToEPICSDataBlockOffset + 2] := #MyWord;
    Else
       #DEVICE_PARAM_OK := FALSE; //Invalid Hash
    END_IF;
END_FUNCTION_BLOCK

DATA_BLOCK "DEV_LEBT-020:ID-IBS-001_iDB"
{ S7_Optimized_Access := 'TRUE' }
VERSION : 1.0
NON_RETAIN
"DEVTYPE_ISRC_LEBT_BDump"
BEGIN
END_DATA_BLOCK


DATA_BLOCK "DEV_LEBT-010:BMD-Chop_iDB"
{ S7_Optimized_Access := 'TRUE' }
VERSION : 1.0
NON_RETAIN
"DEVTYPE_ISRC_LEBT_CHOP"
BEGIN
END_DATA_BLOCK


DATA_BLOCK "DEV_ISrc-010:ISS-Coil-01_iDB"
{ S7_Optimized_Access := 'TRUE' }
VERSION : 1.0
NON_RETAIN
"DEVTYPE_ISRC_LEBT_COIL_SOLENOID"
BEGIN
END_DATA_BLOCK


DATA_BLOCK "DEV_ISrc-010:ISS-Coil-02_iDB"
{ S7_Optimized_Access := 'TRUE' }
VERSION : 1.0
NON_RETAIN
"DEVTYPE_ISRC_LEBT_COIL_SOLENOID"
BEGIN
END_DATA_BLOCK


DATA_BLOCK "DEV_ISrc-010:ISS-Coil-03_iDB"
{ S7_Optimized_Access := 'TRUE' }
VERSION : 1.0
NON_RETAIN
"DEVTYPE_ISRC_LEBT_COIL_SOLENOID"
BEGIN
END_DATA_BLOCK


DATA_BLOCK "DEV_LEBT-010:BMD-Sol-01_iDB"
{ S7_Optimized_Access := 'TRUE' }
VERSION : 1.0
NON_RETAIN
"DEVTYPE_ISRC_LEBT_COIL_SOLENOID"
BEGIN
END_DATA_BLOCK


DATA_BLOCK "DEV_LEBT-010:BMD-Sol-02_iDB"
{ S7_Optimized_Access := 'TRUE' }
VERSION : 1.0
NON_RETAIN
"DEVTYPE_ISRC_LEBT_COIL_SOLENOID"
BEGIN
END_DATA_BLOCK


DATA_BLOCK "DEV_LEBT-010:ID-Coll_iDB"
{ S7_Optimized_Access := 'TRUE' }
VERSION : 1.0
NON_RETAIN
"DEVTYPE_ISRC_LEBT_COLL"
BEGIN
END_DATA_BLOCK


DATA_BLOCK "DEV_ISrc-010:PwrC-HVIT-01_iDB"
{ S7_Optimized_Access := 'TRUE' }
VERSION : 1.0
NON_RETAIN
"DEVTYPE_ISRC_LEBT_HVIT"
BEGIN
END_DATA_BLOCK


DATA_BLOCK "DEV_ISrc-010:ISS-HVPS_iDB"
{ S7_Optimized_Access := 'TRUE' }
VERSION : 1.0
NON_RETAIN
"DEVTYPE_ISRC_LEBT_HVPS"
BEGIN
END_DATA_BLOCK


DATA_BLOCK "DEV_ISrc-010:ISS-HVPf-Doors_iDB"
{ S7_Optimized_Access := 'TRUE' }
VERSION : 1.0
NON_RETAIN
"DEVTYPE_ISRC_LEBT_HVPf_Doors"
BEGIN
END_DATA_BLOCK


DATA_BLOCK "DEV_ISrc-010:ISS-HVPf-Res_iDB"
{ S7_Optimized_Access := 'TRUE' }
VERSION : 1.0
NON_RETAIN
"DEVTYPE_ISRC_LEBT_HVPf_Res"
BEGIN
END_DATA_BLOCK


DATA_BLOCK "DEV_ISrc-010:ISS-Intf-DIAG_iDB"
{ S7_Optimized_Access := 'TRUE' }
VERSION : 1.0
NON_RETAIN
"DEVTYPE_ISRC_LEBT_INTF_DIAG"
BEGIN
END_DATA_BLOCK


DATA_BLOCK "DEV_ISrc-010:ISS-Intf-DPL_iDB"
{ S7_Optimized_Access := 'TRUE' }
VERSION : 1.0
NON_RETAIN
"DEVTYPE_ISRC_LEBT_INTF_DPL"
BEGIN
END_DATA_BLOCK


DATA_BLOCK "DEV_ISrc-010:ISS-Intf-EMU_iDB"
{ S7_Optimized_Access := 'TRUE' }
VERSION : 1.0
NON_RETAIN
"DEVTYPE_ISRC_LEBT_INTF_EMU"
BEGIN
END_DATA_BLOCK


DATA_BLOCK "DEV_ISrc-010:ISS-Intf-HMI_iDB"
{ S7_Optimized_Access := 'TRUE' }
VERSION : 1.0
NON_RETAIN
"DEVTYPE_ISRC_LEBT_INTF_HMI"
BEGIN
END_DATA_BLOCK


DATA_BLOCK "DEV_ISrc-010:ISS-Intf-MPS_iDB"
{ S7_Optimized_Access := 'TRUE' }
VERSION : 1.0
NON_RETAIN
"DEVTYPE_ISRC_LEBT_INTF_MPS"
BEGIN
END_DATA_BLOCK


DATA_BLOCK "DEV_ISrc-010:ISS-Intf-PSS_iDB"
{ S7_Optimized_Access := 'TRUE' }
VERSION : 1.0
NON_RETAIN
"DEVTYPE_ISRC_LEBT_INTF_PSS"
BEGIN
END_DATA_BLOCK


DATA_BLOCK "DEV_ISrc-010:ISS-Intf-Vac_iDB"
{ S7_Optimized_Access := 'TRUE' }
VERSION : 1.0
NON_RETAIN
"DEVTYPE_ISRC_LEBT_INTF_VAC"
BEGIN
END_DATA_BLOCK


DATA_BLOCK "DEV_LEBT-010:ID-Iris_iDB"
{ S7_Optimized_Access := 'TRUE' }
VERSION : 1.0
NON_RETAIN
"DEVTYPE_ISRC_LEBT_IRIS"
BEGIN
END_DATA_BLOCK


DATA_BLOCK "DEV_ISrc-010:ISS-Magtr_iDB"
{ S7_Optimized_Access := 'TRUE' }
VERSION : 1.0
NON_RETAIN
"DEVTYPE_ISRC_LEBT_Magtr"
BEGIN
END_DATA_BLOCK


DATA_BLOCK "DEV_ISrc-010:ISS-MatTr_iDB"
{ S7_Optimized_Access := 'TRUE' }
VERSION : 1.0
NON_RETAIN
"DEVTYPE_ISRC_LEBT_MatTr"
BEGIN
END_DATA_BLOCK


DATA_BLOCK "DEV_LEBT-010:PBI-EMU-001_iDB"
{ S7_Optimized_Access := 'TRUE' }
VERSION : 1.0
NON_RETAIN
"DEVTYPE_ISRC_LEBT_PBI_EMU"
BEGIN
END_DATA_BLOCK


DATA_BLOCK "DEV_LEBT-010:PBI-FC-001_iDB"
{ S7_Optimized_Access := 'TRUE' }
VERSION : 1.0
NON_RETAIN
"DEVTYPE_ISRC_LEBT_PBI_FC"
BEGIN
END_DATA_BLOCK


DATA_BLOCK "DEV_ISrc-010:PwrC-CoilPS-01_iDB"
{ S7_Optimized_Access := 'TRUE' }
VERSION : 1.0
NON_RETAIN
"DEVTYPE_ISRC_LEBT_PS_COIL"
BEGIN
END_DATA_BLOCK


DATA_BLOCK "DEV_ISrc-010:PwrC-CoilPS-02_iDB"
{ S7_Optimized_Access := 'TRUE' }
VERSION : 1.0
NON_RETAIN
"DEVTYPE_ISRC_LEBT_PS_COIL"
BEGIN
END_DATA_BLOCK


DATA_BLOCK "DEV_ISrc-010:PwrC-CoilPS-03_iDB"
{ S7_Optimized_Access := 'TRUE' }
VERSION : 1.0
NON_RETAIN
"DEVTYPE_ISRC_LEBT_PS_COIL"
BEGIN
END_DATA_BLOCK


DATA_BLOCK "DEV_ISrc-010:PwrC-RepPS-01_iDB"
{ S7_Optimized_Access := 'TRUE' }
VERSION : 1.0
NON_RETAIN
"DEVTYPE_ISRC_LEBT_PS_REP"
BEGIN
END_DATA_BLOCK


DATA_BLOCK "DEV_LEBT-010:PwrC-RepPS-01_iDB"
{ S7_Optimized_Access := 'TRUE' }
VERSION : 1.0
NON_RETAIN
"DEVTYPE_ISRC_LEBT_PS_REP"
BEGIN
END_DATA_BLOCK


DATA_BLOCK "DEV_LEBT-010:PwrC-PSCH-01_iDB"
{ S7_Optimized_Access := 'TRUE' }
VERSION : 1.0
NON_RETAIN
"DEVTYPE_ISRC_LEBT_PS_SOL_STR"
BEGIN
END_DATA_BLOCK


DATA_BLOCK "DEV_LEBT-010:PwrC-PSCH-02_iDB"
{ S7_Optimized_Access := 'TRUE' }
VERSION : 1.0
NON_RETAIN
"DEVTYPE_ISRC_LEBT_PS_SOL_STR"
BEGIN
END_DATA_BLOCK


DATA_BLOCK "DEV_LEBT-010:PwrC-PSCV-01_iDB"
{ S7_Optimized_Access := 'TRUE' }
VERSION : 1.0
NON_RETAIN
"DEVTYPE_ISRC_LEBT_PS_SOL_STR"
BEGIN
END_DATA_BLOCK


DATA_BLOCK "DEV_LEBT-010:PwrC-PSCV-02_iDB"
{ S7_Optimized_Access := 'TRUE' }
VERSION : 1.0
NON_RETAIN
"DEVTYPE_ISRC_LEBT_PS_SOL_STR"
BEGIN
END_DATA_BLOCK


DATA_BLOCK "DEV_LEBT-010:PwrC-SolPS-01_iDB"
{ S7_Optimized_Access := 'TRUE' }
VERSION : 1.0
NON_RETAIN
"DEVTYPE_ISRC_LEBT_PS_SOL_STR"
BEGIN
END_DATA_BLOCK


DATA_BLOCK "DEV_LEBT-010:PwrC-SolPS-02_iDB"
{ S7_Optimized_Access := 'TRUE' }
VERSION : 1.0
NON_RETAIN
"DEVTYPE_ISRC_LEBT_PS_SOL_STR"
BEGIN
END_DATA_BLOCK


DATA_BLOCK "DEV_ISrc-010:ISS-PlasCh_iDB"
{ S7_Optimized_Access := 'TRUE' }
VERSION : 1.0
NON_RETAIN
"DEVTYPE_ISRC_LEBT_PlasCh"
BEGIN
END_DATA_BLOCK


DATA_BLOCK "DEV_ISrc-010:BMD-Rep-01_iDB"
{ S7_Optimized_Access := 'TRUE' }
VERSION : 1.0
NON_RETAIN
"DEVTYPE_ISRC_LEBT_REP"
BEGIN
END_DATA_BLOCK


DATA_BLOCK "DEV_LEBT-010:BMD-CH-01_iDB"
{ S7_Optimized_Access := 'TRUE' }
VERSION : 1.0
NON_RETAIN
"DEVTYPE_ISRC_LEBT_STR"
BEGIN
END_DATA_BLOCK


DATA_BLOCK "DEV_LEBT-010:BMD-CH-02_iDB"
{ S7_Optimized_Access := 'TRUE' }
VERSION : 1.0
NON_RETAIN
"DEVTYPE_ISRC_LEBT_STR"
BEGIN
END_DATA_BLOCK


DATA_BLOCK "DEV_LEBT-010:BMD-CV-01_iDB"
{ S7_Optimized_Access := 'TRUE' }
VERSION : 1.0
NON_RETAIN
"DEVTYPE_ISRC_LEBT_STR"
BEGIN
END_DATA_BLOCK


DATA_BLOCK "DEV_LEBT-010:BMD-CV-02_iDB"
{ S7_Optimized_Access := 'TRUE' }
VERSION : 1.0
NON_RETAIN
"DEVTYPE_ISRC_LEBT_STR"
BEGIN
END_DATA_BLOCK


DATA_BLOCK "DEV_ISrc-010:Vac-VVA-01100_iDB"
{ S7_Optimized_Access := 'TRUE' }
VERSION : 1.0
NON_RETAIN
"DEVTYPE_ISRC_LEBT_VAC_VVA"
BEGIN
END_DATA_BLOCK


DATA_BLOCK "DEV_ISrc-010:WtrC-PT-001_iDB"
{ S7_Optimized_Access := 'TRUE' }
VERSION : 1.0
NON_RETAIN
"DEVTYPE_ISRC_LEBT_WTRC_PRES"
BEGIN
END_DATA_BLOCK


DATA_BLOCK "DEV_ISrc-010:WtrC-PT-002_iDB"
{ S7_Optimized_Access := 'TRUE' }
VERSION : 1.0
NON_RETAIN
"DEVTYPE_ISRC_LEBT_WTRC_PRES"
BEGIN
END_DATA_BLOCK


DATA_BLOCK "DEV_ISrc-010:WtrC-PT-011_iDB"
{ S7_Optimized_Access := 'TRUE' }
VERSION : 1.0
NON_RETAIN
"DEVTYPE_ISRC_LEBT_WTRC_PRES"
BEGIN
END_DATA_BLOCK


DATA_BLOCK "DEV_ISrc-010:WtrC-PT-012_iDB"
{ S7_Optimized_Access := 'TRUE' }
VERSION : 1.0
NON_RETAIN
"DEVTYPE_ISRC_LEBT_WTRC_PRES"
BEGIN
END_DATA_BLOCK


DATA_BLOCK "DEV_ISrc-010:WtrC-TT-001_iDB"
{ S7_Optimized_Access := 'TRUE' }
VERSION : 1.0
NON_RETAIN
"DEVTYPE_ISRC_LEBT_WTRC_TEMP"
BEGIN
END_DATA_BLOCK


DATA_BLOCK "DEV_ISrc-010:WtrC-TT-011_iDB"
{ S7_Optimized_Access := 'TRUE' }
VERSION : 1.0
NON_RETAIN
"DEVTYPE_ISRC_LEBT_WTRC_TEMP"
BEGIN
END_DATA_BLOCK


DATA_BLOCK "DEV_ISrc-010:WtrC-TT-012_iDB"
{ S7_Optimized_Access := 'TRUE' }
VERSION : 1.0
NON_RETAIN
"DEVTYPE_ISRC_LEBT_WTRC_TEMP"
BEGIN
END_DATA_BLOCK

FUNCTION "EPICS_device_calls" : Void
{ S7_Optimized_Access := 'TRUE' }
VERSION : 1.0

   VAR_TEMP
      "LEBT-020:ID-IBS-001" : Bool;   // HASH codes are OK
      "LEBT-010:BMD-Chop" : Bool;   // HASH codes are OK
      "ISrc-010:ISS-Coil-01" : Bool;   // HASH codes are OK
      "ISrc-010:ISS-Coil-02" : Bool;   // HASH codes are OK
      "ISrc-010:ISS-Coil-03" : Bool;   // HASH codes are OK
      "LEBT-010:BMD-Sol-01" : Bool;   // HASH codes are OK
      "LEBT-010:BMD-Sol-02" : Bool;   // HASH codes are OK
      "LEBT-010:ID-Coll" : Bool;   // HASH codes are OK
      "ISrc-010:PwrC-HVIT-01" : Bool;   // HASH codes are OK
      "ISrc-010:ISS-HVPS" : Bool;   // HASH codes are OK
      "ISrc-010:ISS-HVPf-Doors" : Bool;   // HASH codes are OK
      "ISrc-010:ISS-HVPf-Res" : Bool;   // HASH codes are OK
      "ISrc-010:ISS-Intf-DIAG" : Bool;   // HASH codes are OK
      "ISrc-010:ISS-Intf-DPL" : Bool;   // HASH codes are OK
      "ISrc-010:ISS-Intf-EMU" : Bool;   // HASH codes are OK
      "ISrc-010:ISS-Intf-HMI" : Bool;   // HASH codes are OK
      "ISrc-010:ISS-Intf-MPS" : Bool;   // HASH codes are OK
      "ISrc-010:ISS-Intf-PSS" : Bool;   // HASH codes are OK
      "ISrc-010:ISS-Intf-Vac" : Bool;   // HASH codes are OK
      "LEBT-010:ID-Iris" : Bool;   // HASH codes are OK
      "ISrc-010:ISS-Magtr" : Bool;   // HASH codes are OK
      "ISrc-010:ISS-MatTr" : Bool;   // HASH codes are OK
      "LEBT-010:PBI-EMU-001" : Bool;   // HASH codes are OK
      "LEBT-010:PBI-FC-001" : Bool;   // HASH codes are OK
      "ISrc-010:PwrC-CoilPS-01" : Bool;   // HASH codes are OK
      "ISrc-010:PwrC-CoilPS-02" : Bool;   // HASH codes are OK
      "ISrc-010:PwrC-CoilPS-03" : Bool;   // HASH codes are OK
      "ISrc-010:PwrC-RepPS-01" : Bool;   // HASH codes are OK
      "LEBT-010:PwrC-RepPS-01" : Bool;   // HASH codes are OK
      "LEBT-010:PwrC-PSCH-01" : Bool;   // HASH codes are OK
      "LEBT-010:PwrC-PSCH-02" : Bool;   // HASH codes are OK
      "LEBT-010:PwrC-PSCV-01" : Bool;   // HASH codes are OK
      "LEBT-010:PwrC-PSCV-02" : Bool;   // HASH codes are OK
      "LEBT-010:PwrC-SolPS-01" : Bool;   // HASH codes are OK
      "LEBT-010:PwrC-SolPS-02" : Bool;   // HASH codes are OK
      "ISrc-010:ISS-PlasCh" : Bool;   // HASH codes are OK
      "ISrc-010:BMD-Rep-01" : Bool;   // HASH codes are OK
      "LEBT-010:BMD-CH-01" : Bool;   // HASH codes are OK
      "LEBT-010:BMD-CH-02" : Bool;   // HASH codes are OK
      "LEBT-010:BMD-CV-01" : Bool;   // HASH codes are OK
      "LEBT-010:BMD-CV-02" : Bool;   // HASH codes are OK
      "ISrc-010:Vac-VVA-01100" : Bool;   // HASH codes are OK
      "ISrc-010:WtrC-PT-001" : Bool;   // HASH codes are OK
      "ISrc-010:WtrC-PT-002" : Bool;   // HASH codes are OK
      "ISrc-010:WtrC-PT-011" : Bool;   // HASH codes are OK
      "ISrc-010:WtrC-PT-012" : Bool;   // HASH codes are OK
      "ISrc-010:WtrC-TT-001" : Bool;   // HASH codes are OK
      "ISrc-010:WtrC-TT-011" : Bool;   // HASH codes are OK
      "ISrc-010:WtrC-TT-012" : Bool;   // HASH codes are OK
   END_VAR

BEGIN
      //Author: Miklos Boros (miklos.boros@esss.se), Copyrigth 2017-2019 by European Spallation Source, Lund
      //This block was generated by PLCFactory
      //According to HASH:1347332123
      //Description: Description: This function calls the devices according to the corresponding device type

        //DO NOT Modify the following line!!!
        "Utilities".TestInProgress := FALSE;
        "Utilities".EPICS_Device_calls_precessed := TRUE;


        //********************************************
        // Device name: LEBT-020:ID-IBS-001
        // Device type: ISRC_LEBT_BDump
        //********************************************

      "DEV_LEBT-020:ID-IBS-001_iDB" (EPICSToPLCLength:=0,
      EPICSToPLCDataBlockOffset:=0+10,
      EPICSToPLCParametersStart:=0,
      PLCToEPICSLength:=1,
      PLCToEPICSDataBlockOffset:=0+10);

        //********************************************
        // Device name: LEBT-010:BMD-Chop
        // Device type: ISRC_LEBT_CHOP
        //********************************************

      "DEV_LEBT-010:BMD-Chop_iDB" (EPICSToPLCLength:=1,
      EPICSToPLCDataBlockOffset:=0+10,
      EPICSToPLCParametersStart:=1,
      PLCToEPICSLength:=1,
      PLCToEPICSDataBlockOffset:=1+10);

        //********************************************
        // Device name: ISrc-010:ISS-Coil-01
        // Device type: ISRC_LEBT_COIL_SOLENOID
        //********************************************

      "DEV_ISrc-010:ISS-Coil-01_iDB" (EPICSToPLCLength:=0,
      EPICSToPLCDataBlockOffset:=1+10,
      EPICSToPLCParametersStart:=0,
      PLCToEPICSLength:=1,
      PLCToEPICSDataBlockOffset:=2+10);

        //********************************************
        // Device name: ISrc-010:ISS-Coil-02
        // Device type: ISRC_LEBT_COIL_SOLENOID
        //********************************************

      "DEV_ISrc-010:ISS-Coil-02_iDB" (EPICSToPLCLength:=0,
      EPICSToPLCDataBlockOffset:=1+10,
      EPICSToPLCParametersStart:=0,
      PLCToEPICSLength:=1,
      PLCToEPICSDataBlockOffset:=3+10);

        //********************************************
        // Device name: ISrc-010:ISS-Coil-03
        // Device type: ISRC_LEBT_COIL_SOLENOID
        //********************************************

      "DEV_ISrc-010:ISS-Coil-03_iDB" (EPICSToPLCLength:=0,
      EPICSToPLCDataBlockOffset:=1+10,
      EPICSToPLCParametersStart:=0,
      PLCToEPICSLength:=1,
      PLCToEPICSDataBlockOffset:=4+10);

        //********************************************
        // Device name: LEBT-010:BMD-Sol-01
        // Device type: ISRC_LEBT_COIL_SOLENOID
        //********************************************

      "DEV_LEBT-010:BMD-Sol-01_iDB" (EPICSToPLCLength:=0,
      EPICSToPLCDataBlockOffset:=1+10,
      EPICSToPLCParametersStart:=0,
      PLCToEPICSLength:=1,
      PLCToEPICSDataBlockOffset:=5+10);

        //********************************************
        // Device name: LEBT-010:BMD-Sol-02
        // Device type: ISRC_LEBT_COIL_SOLENOID
        //********************************************

      "DEV_LEBT-010:BMD-Sol-02_iDB" (EPICSToPLCLength:=0,
      EPICSToPLCDataBlockOffset:=1+10,
      EPICSToPLCParametersStart:=0,
      PLCToEPICSLength:=1,
      PLCToEPICSDataBlockOffset:=6+10);

        //********************************************
        // Device name: LEBT-010:ID-Coll
        // Device type: ISRC_LEBT_COLL
        //********************************************

      "DEV_LEBT-010:ID-Coll_iDB" (EPICSToPLCLength:=0,
      EPICSToPLCDataBlockOffset:=1+10,
      EPICSToPLCParametersStart:=0,
      PLCToEPICSLength:=1,
      PLCToEPICSDataBlockOffset:=7+10);

        //********************************************
        // Device name: ISrc-010:PwrC-HVIT-01
        // Device type: ISRC_LEBT_HVIT
        //********************************************

      "DEV_ISrc-010:PwrC-HVIT-01_iDB" (EPICSToPLCLength:=0,
      EPICSToPLCDataBlockOffset:=1+10,
      EPICSToPLCParametersStart:=0,
      PLCToEPICSLength:=1,
      PLCToEPICSDataBlockOffset:=8+10);

        //********************************************
        // Device name: ISrc-010:ISS-HVPS
        // Device type: ISRC_LEBT_HVPS
        //********************************************

      "DEV_ISrc-010:ISS-HVPS_iDB" (EPICSToPLCLength:=4,
      EPICSToPLCDataBlockOffset:=1+10,
      EPICSToPLCParametersStart:=1,
      PLCToEPICSLength:=1,
      PLCToEPICSDataBlockOffset:=9+10);

        //********************************************
        // Device name: ISrc-010:ISS-HVPf-Doors
        // Device type: ISRC_LEBT_HVPf_Doors
        //********************************************

      "DEV_ISrc-010:ISS-HVPf-Doors_iDB" (EPICSToPLCLength:=0,
      EPICSToPLCDataBlockOffset:=5+10,
      EPICSToPLCParametersStart:=0,
      PLCToEPICSLength:=1,
      PLCToEPICSDataBlockOffset:=10+10);

        //********************************************
        // Device name: ISrc-010:ISS-HVPf-Res
        // Device type: ISRC_LEBT_HVPf_Res
        //********************************************

      "DEV_ISrc-010:ISS-HVPf-Res_iDB" (EPICSToPLCLength:=0,
      EPICSToPLCDataBlockOffset:=5+10,
      EPICSToPLCParametersStart:=0,
      PLCToEPICSLength:=1,
      PLCToEPICSDataBlockOffset:=11+10);

        //********************************************
        // Device name: ISrc-010:ISS-Intf-DIAG
        // Device type: ISRC_LEBT_INTF_DIAG
        //********************************************

      "DEV_ISrc-010:ISS-Intf-DIAG_iDB" (EPICSToPLCLength:=0,
      EPICSToPLCDataBlockOffset:=5+10,
      EPICSToPLCParametersStart:=0,
      PLCToEPICSLength:=2,
      PLCToEPICSDataBlockOffset:=12+10);

        //********************************************
        // Device name: ISrc-010:ISS-Intf-DPL
        // Device type: ISRC_LEBT_INTF_DPL
        //********************************************

      "DEV_ISrc-010:ISS-Intf-DPL_iDB" (EPICSToPLCLength:=0,
      EPICSToPLCDataBlockOffset:=5+10,
      EPICSToPLCParametersStart:=0,
      PLCToEPICSLength:=1,
      PLCToEPICSDataBlockOffset:=14+10);

        //********************************************
        // Device name: ISrc-010:ISS-Intf-EMU
        // Device type: ISRC_LEBT_INTF_EMU
        //********************************************

      "DEV_ISrc-010:ISS-Intf-EMU_iDB" (EPICSToPLCLength:=0,
      EPICSToPLCDataBlockOffset:=5+10,
      EPICSToPLCParametersStart:=0,
      PLCToEPICSLength:=1,
      PLCToEPICSDataBlockOffset:=15+10);

        //********************************************
        // Device name: ISrc-010:ISS-Intf-HMI
        // Device type: ISRC_LEBT_INTF_HMI
        //********************************************

      "DEV_ISrc-010:ISS-Intf-HMI_iDB" (EPICSToPLCLength:=3,
      EPICSToPLCDataBlockOffset:=5+10,
      EPICSToPLCParametersStart:=1,
      PLCToEPICSLength:=9,
      PLCToEPICSDataBlockOffset:=16+10);

        //********************************************
        // Device name: ISrc-010:ISS-Intf-MPS
        // Device type: ISRC_LEBT_INTF_MPS
        //********************************************

      "DEV_ISrc-010:ISS-Intf-MPS_iDB" (EPICSToPLCLength:=0,
      EPICSToPLCDataBlockOffset:=8+10,
      EPICSToPLCParametersStart:=0,
      PLCToEPICSLength:=1,
      PLCToEPICSDataBlockOffset:=25+10);

        //********************************************
        // Device name: ISrc-010:ISS-Intf-PSS
        // Device type: ISRC_LEBT_INTF_PSS
        //********************************************

      "DEV_ISrc-010:ISS-Intf-PSS_iDB" (EPICSToPLCLength:=0,
      EPICSToPLCDataBlockOffset:=8+10,
      EPICSToPLCParametersStart:=0,
      PLCToEPICSLength:=1,
      PLCToEPICSDataBlockOffset:=26+10);

        //********************************************
        // Device name: ISrc-010:ISS-Intf-Vac
        // Device type: ISRC_LEBT_INTF_VAC
        //********************************************

      "DEV_ISrc-010:ISS-Intf-Vac_iDB" (EPICSToPLCLength:=0,
      EPICSToPLCDataBlockOffset:=8+10,
      EPICSToPLCParametersStart:=0,
      PLCToEPICSLength:=1,
      PLCToEPICSDataBlockOffset:=27+10);

        //********************************************
        // Device name: LEBT-010:ID-Iris
        // Device type: ISRC_LEBT_IRIS
        //********************************************

      "DEV_LEBT-010:ID-Iris_iDB" (EPICSToPLCLength:=0,
      EPICSToPLCDataBlockOffset:=8+10,
      EPICSToPLCParametersStart:=0,
      PLCToEPICSLength:=1,
      PLCToEPICSDataBlockOffset:=28+10);

        //********************************************
        // Device name: ISrc-010:ISS-Magtr
        // Device type: ISRC_LEBT_Magtr
        //********************************************

      "DEV_ISrc-010:ISS-Magtr_iDB" (EPICSToPLCLength:=1,
      EPICSToPLCDataBlockOffset:=8+10,
      EPICSToPLCParametersStart:=0,
      PLCToEPICSLength:=1,
      PLCToEPICSDataBlockOffset:=29+10);

        //********************************************
        // Device name: ISrc-010:ISS-MatTr
        // Device type: ISRC_LEBT_MatTr
        //********************************************

      "DEV_ISrc-010:ISS-MatTr_iDB" (EPICSToPLCLength:=0,
      EPICSToPLCDataBlockOffset:=9+10,
      EPICSToPLCParametersStart:=0,
      PLCToEPICSLength:=1,
      PLCToEPICSDataBlockOffset:=30+10);

        //********************************************
        // Device name: LEBT-010:PBI-EMU-001
        // Device type: ISRC_LEBT_PBI_EMU
        //********************************************

      "DEV_LEBT-010:PBI-EMU-001_iDB" (EPICSToPLCLength:=0,
      EPICSToPLCDataBlockOffset:=9+10,
      EPICSToPLCParametersStart:=0,
      PLCToEPICSLength:=1,
      PLCToEPICSDataBlockOffset:=31+10);

        //********************************************
        // Device name: LEBT-010:PBI-FC-001
        // Device type: ISRC_LEBT_PBI_FC
        //********************************************

      "DEV_LEBT-010:PBI-FC-001_iDB" (EPICSToPLCLength:=0,
      EPICSToPLCDataBlockOffset:=9+10,
      EPICSToPLCParametersStart:=0,
      PLCToEPICSLength:=1,
      PLCToEPICSDataBlockOffset:=32+10);

        //********************************************
        // Device name: ISrc-010:PwrC-CoilPS-01
        // Device type: ISRC_LEBT_PS_COIL
        //********************************************

      "DEV_ISrc-010:PwrC-CoilPS-01_iDB" (EPICSToPLCLength:=0,
      EPICSToPLCDataBlockOffset:=9+10,
      EPICSToPLCParametersStart:=0,
      PLCToEPICSLength:=1,
      PLCToEPICSDataBlockOffset:=33+10);

        //********************************************
        // Device name: ISrc-010:PwrC-CoilPS-02
        // Device type: ISRC_LEBT_PS_COIL
        //********************************************

      "DEV_ISrc-010:PwrC-CoilPS-02_iDB" (EPICSToPLCLength:=0,
      EPICSToPLCDataBlockOffset:=9+10,
      EPICSToPLCParametersStart:=0,
      PLCToEPICSLength:=1,
      PLCToEPICSDataBlockOffset:=34+10);

        //********************************************
        // Device name: ISrc-010:PwrC-CoilPS-03
        // Device type: ISRC_LEBT_PS_COIL
        //********************************************

      "DEV_ISrc-010:PwrC-CoilPS-03_iDB" (EPICSToPLCLength:=0,
      EPICSToPLCDataBlockOffset:=9+10,
      EPICSToPLCParametersStart:=0,
      PLCToEPICSLength:=1,
      PLCToEPICSDataBlockOffset:=35+10);

        //********************************************
        // Device name: ISrc-010:PwrC-RepPS-01
        // Device type: ISRC_LEBT_PS_REP
        //********************************************

      "DEV_ISrc-010:PwrC-RepPS-01_iDB" (EPICSToPLCLength:=2,
      EPICSToPLCDataBlockOffset:=9+10,
      EPICSToPLCParametersStart:=0,
      PLCToEPICSLength:=1,
      PLCToEPICSDataBlockOffset:=36+10);

        //********************************************
        // Device name: LEBT-010:PwrC-RepPS-01
        // Device type: ISRC_LEBT_PS_REP
        //********************************************

      "DEV_LEBT-010:PwrC-RepPS-01_iDB" (EPICSToPLCLength:=2,
      EPICSToPLCDataBlockOffset:=11+10,
      EPICSToPLCParametersStart:=0,
      PLCToEPICSLength:=1,
      PLCToEPICSDataBlockOffset:=37+10);

        //********************************************
        // Device name: LEBT-010:PwrC-PSCH-01
        // Device type: ISRC_LEBT_PS_SOL_STR
        //********************************************

      "DEV_LEBT-010:PwrC-PSCH-01_iDB" (EPICSToPLCLength:=0,
      EPICSToPLCDataBlockOffset:=13+10,
      EPICSToPLCParametersStart:=0,
      PLCToEPICSLength:=3,
      PLCToEPICSDataBlockOffset:=38+10);

        //********************************************
        // Device name: LEBT-010:PwrC-PSCH-02
        // Device type: ISRC_LEBT_PS_SOL_STR
        //********************************************

      "DEV_LEBT-010:PwrC-PSCH-02_iDB" (EPICSToPLCLength:=0,
      EPICSToPLCDataBlockOffset:=13+10,
      EPICSToPLCParametersStart:=0,
      PLCToEPICSLength:=3,
      PLCToEPICSDataBlockOffset:=41+10);

        //********************************************
        // Device name: LEBT-010:PwrC-PSCV-01
        // Device type: ISRC_LEBT_PS_SOL_STR
        //********************************************

      "DEV_LEBT-010:PwrC-PSCV-01_iDB" (EPICSToPLCLength:=0,
      EPICSToPLCDataBlockOffset:=13+10,
      EPICSToPLCParametersStart:=0,
      PLCToEPICSLength:=3,
      PLCToEPICSDataBlockOffset:=44+10);

        //********************************************
        // Device name: LEBT-010:PwrC-PSCV-02
        // Device type: ISRC_LEBT_PS_SOL_STR
        //********************************************

      "DEV_LEBT-010:PwrC-PSCV-02_iDB" (EPICSToPLCLength:=0,
      EPICSToPLCDataBlockOffset:=13+10,
      EPICSToPLCParametersStart:=0,
      PLCToEPICSLength:=3,
      PLCToEPICSDataBlockOffset:=47+10);

        //********************************************
        // Device name: LEBT-010:PwrC-SolPS-01
        // Device type: ISRC_LEBT_PS_SOL_STR
        //********************************************

      "DEV_LEBT-010:PwrC-SolPS-01_iDB" (EPICSToPLCLength:=0,
      EPICSToPLCDataBlockOffset:=13+10,
      EPICSToPLCParametersStart:=0,
      PLCToEPICSLength:=3,
      PLCToEPICSDataBlockOffset:=50+10);

        //********************************************
        // Device name: LEBT-010:PwrC-SolPS-02
        // Device type: ISRC_LEBT_PS_SOL_STR
        //********************************************

      "DEV_LEBT-010:PwrC-SolPS-02_iDB" (EPICSToPLCLength:=0,
      EPICSToPLCDataBlockOffset:=13+10,
      EPICSToPLCParametersStart:=0,
      PLCToEPICSLength:=3,
      PLCToEPICSDataBlockOffset:=53+10);

        //********************************************
        // Device name: ISrc-010:ISS-PlasCh
        // Device type: ISRC_LEBT_PlasCh
        //********************************************

      "DEV_ISrc-010:ISS-PlasCh_iDB" (EPICSToPLCLength:=0,
      EPICSToPLCDataBlockOffset:=13+10,
      EPICSToPLCParametersStart:=0,
      PLCToEPICSLength:=1,
      PLCToEPICSDataBlockOffset:=56+10);

        //********************************************
        // Device name: ISrc-010:BMD-Rep-01
        // Device type: ISRC_LEBT_REP
        //********************************************

      "DEV_ISrc-010:BMD-Rep-01_iDB" (EPICSToPLCLength:=0,
      EPICSToPLCDataBlockOffset:=13+10,
      EPICSToPLCParametersStart:=0,
      PLCToEPICSLength:=1,
      PLCToEPICSDataBlockOffset:=57+10);

        //********************************************
        // Device name: LEBT-010:BMD-CH-01
        // Device type: ISRC_LEBT_STR
        //********************************************

      "DEV_LEBT-010:BMD-CH-01_iDB" (EPICSToPLCLength:=1,
      EPICSToPLCDataBlockOffset:=13+10,
      EPICSToPLCParametersStart:=1,
      PLCToEPICSLength:=1,
      PLCToEPICSDataBlockOffset:=58+10);

        //********************************************
        // Device name: LEBT-010:BMD-CH-02
        // Device type: ISRC_LEBT_STR
        //********************************************

      "DEV_LEBT-010:BMD-CH-02_iDB" (EPICSToPLCLength:=1,
      EPICSToPLCDataBlockOffset:=14+10,
      EPICSToPLCParametersStart:=1,
      PLCToEPICSLength:=1,
      PLCToEPICSDataBlockOffset:=59+10);

        //********************************************
        // Device name: LEBT-010:BMD-CV-01
        // Device type: ISRC_LEBT_STR
        //********************************************

      "DEV_LEBT-010:BMD-CV-01_iDB" (EPICSToPLCLength:=1,
      EPICSToPLCDataBlockOffset:=15+10,
      EPICSToPLCParametersStart:=1,
      PLCToEPICSLength:=1,
      PLCToEPICSDataBlockOffset:=60+10);

        //********************************************
        // Device name: LEBT-010:BMD-CV-02
        // Device type: ISRC_LEBT_STR
        //********************************************

      "DEV_LEBT-010:BMD-CV-02_iDB" (EPICSToPLCLength:=1,
      EPICSToPLCDataBlockOffset:=16+10,
      EPICSToPLCParametersStart:=1,
      PLCToEPICSLength:=1,
      PLCToEPICSDataBlockOffset:=61+10);

        //********************************************
        // Device name: ISrc-010:Vac-VVA-01100
        // Device type: ISRC_LEBT_VAC_VVA
        //********************************************

      "DEV_ISrc-010:Vac-VVA-01100_iDB" (EPICSToPLCLength:=1,
      EPICSToPLCDataBlockOffset:=17+10,
      EPICSToPLCParametersStart:=1,
      PLCToEPICSLength:=1,
      PLCToEPICSDataBlockOffset:=62+10);

        //********************************************
        // Device name: ISrc-010:WtrC-PT-001
        // Device type: ISRC_LEBT_WTRC_PRES
        //********************************************

      "DEV_ISrc-010:WtrC-PT-001_iDB" (EPICSToPLCLength:=0,
      EPICSToPLCDataBlockOffset:=18+10,
      EPICSToPLCParametersStart:=0,
      PLCToEPICSLength:=2,
      PLCToEPICSDataBlockOffset:=63+10);

        //********************************************
        // Device name: ISrc-010:WtrC-PT-002
        // Device type: ISRC_LEBT_WTRC_PRES
        //********************************************

      "DEV_ISrc-010:WtrC-PT-002_iDB" (EPICSToPLCLength:=0,
      EPICSToPLCDataBlockOffset:=18+10,
      EPICSToPLCParametersStart:=0,
      PLCToEPICSLength:=2,
      PLCToEPICSDataBlockOffset:=65+10);

        //********************************************
        // Device name: ISrc-010:WtrC-PT-011
        // Device type: ISRC_LEBT_WTRC_PRES
        //********************************************

      "DEV_ISrc-010:WtrC-PT-011_iDB" (EPICSToPLCLength:=0,
      EPICSToPLCDataBlockOffset:=18+10,
      EPICSToPLCParametersStart:=0,
      PLCToEPICSLength:=2,
      PLCToEPICSDataBlockOffset:=67+10);

        //********************************************
        // Device name: ISrc-010:WtrC-PT-012
        // Device type: ISRC_LEBT_WTRC_PRES
        //********************************************

      "DEV_ISrc-010:WtrC-PT-012_iDB" (EPICSToPLCLength:=0,
      EPICSToPLCDataBlockOffset:=18+10,
      EPICSToPLCParametersStart:=0,
      PLCToEPICSLength:=2,
      PLCToEPICSDataBlockOffset:=69+10);

        //********************************************
        // Device name: ISrc-010:WtrC-TT-001
        // Device type: ISRC_LEBT_WTRC_TEMP
        //********************************************

      "DEV_ISrc-010:WtrC-TT-001_iDB" (EPICSToPLCLength:=0,
      EPICSToPLCDataBlockOffset:=18+10,
      EPICSToPLCParametersStart:=0,
      PLCToEPICSLength:=3,
      PLCToEPICSDataBlockOffset:=71+10);

        //********************************************
        // Device name: ISrc-010:WtrC-TT-011
        // Device type: ISRC_LEBT_WTRC_TEMP
        //********************************************

      "DEV_ISrc-010:WtrC-TT-011_iDB" (EPICSToPLCLength:=0,
      EPICSToPLCDataBlockOffset:=18+10,
      EPICSToPLCParametersStart:=0,
      PLCToEPICSLength:=3,
      PLCToEPICSDataBlockOffset:=74+10);

        //********************************************
        // Device name: ISrc-010:WtrC-TT-012
        // Device type: ISRC_LEBT_WTRC_TEMP
        //********************************************

      "DEV_ISrc-010:WtrC-TT-012_iDB" (EPICSToPLCLength:=0,
      EPICSToPLCDataBlockOffset:=18+10,
      EPICSToPLCParametersStart:=0,
      PLCToEPICSLength:=3,
      PLCToEPICSDataBlockOffset:=77+10);
END_FUNCTION
DATA_BLOCK "EPICS_DebuggerResult"
{ S7_Optimized_Access := 'TRUE' }
VERSION : 0.1
NON_RETAIN
   VAR
      EPICS_Debugger_Checksum : Array[0..7] of Byte;   // Current TIA Portal Software Hash including PLC logic (this is not the EPICS IOC Hash)
      EPICS_Debugger_UtilitiesCall : String;   // PLCFactory Utilities call status
      EPICS_Debugger_DeviceCalls : String;   // PLCFactory DeviceCalls status
      EPICS_Debugger_IOCHash : String;   // EPICS IOC Hash vs. PLCFactory Hash
      EPICS_Debugger_ModBusHeartBeat : String;   // EPICS IOC Modbus (IOC->PLC) communication status
      EPICS_Debugger_S7Connection : String;   // EPICS IOC S7 TCP (PLC->IOC) communication status
      EPICS_Debugger_EPICS_GeneralState : String;   // Main status of the EPICS IOC communication
      EPICS_S7Port : Int;   // Actual TCP port that has been opened by the PLC
      EPICS_ModbusPort : Int;   // Actual ModBusTCP port that has been opened by the PLC
      EPICS_PLC_EthernetInterface : UInt;   // The currently used HW Identifer of the Ethernet Port on the PLC dedicated to EPICS
   END_VAR

BEGIN

END_DATA_BLOCK
FUNCTION_BLOCK "EPICS_DebuggerFB"
{ S7_Optimized_Access := 'TRUE' }
VERSION : 0.1
   VAR
      GetChecksum_Instance {OriginalPartName := 'GetChecksum_FB_807_S71500'; LibVersion := '1.0'; ExternalAccessible := 'False'; ExternalVisible := 'False'; ExternalWritable := 'False'} : GetChecksum;
      execute { ExternalAccessible := 'False'; ExternalVisible := 'False'; ExternalWritable := 'False'} : Bool;
      scope { ExternalAccessible := 'False'; ExternalVisible := 'False'; ExternalWritable := 'False'} : UInt := 1;
      busy { ExternalAccessible := 'False'; ExternalVisible := 'False'; ExternalWritable := 'False'} : Bool;
      done { ExternalAccessible := 'False'; ExternalVisible := 'False'; ExternalWritable := 'False'} : Bool;
      error { ExternalAccessible := 'False'; ExternalVisible := 'False'; ExternalWritable := 'False'} : Bool;
      memErrStatus { ExternalAccessible := 'False'; ExternalVisible := 'False'; ExternalWritable := 'False'} : Word;
      CheckUtilitiesTON {OriginalPartName := 'IEC_TIMER'; LibVersion := '1.0'; ExternalAccessible := 'False'; ExternalVisible := 'False'; ExternalWritable := 'False'} : TON_TIME;
      UtilSquareErrorTON { ExternalAccessible := 'False'; ExternalVisible := 'False'; ExternalWritable := 'False'} : Bool;
      CheckUtilitiesTON2 {OriginalPartName := 'IEC_TIMER'; LibVersion := '1.0'; ExternalAccessible := 'False'; ExternalVisible := 'False'; ExternalWritable := 'False'} : TON_TIME;
      UtilSquareErrorTON2 { ExternalAccessible := 'False'; ExternalVisible := 'False'; ExternalWritable := 'False'} : Bool;
      ModBus_TON {OriginalPartName := 'IEC_TIMER'; LibVersion := '1.0'; ExternalAccessible := 'False'; ExternalVisible := 'False'; ExternalWritable := 'False'} : TON_TIME;
      ModBus_wordsave { ExternalAccessible := 'False'; ExternalVisible := 'False'; ExternalWritable := 'False'} : Word;
   END_VAR
   VAR DB_SPECIFIC
      Helper_String { ExternalAccessible := 'False'; ExternalVisible := 'False'; ExternalWritable := 'False'} : String;
      Helper_String_Array { ExternalAccessible := 'False'; ExternalVisible := 'False'; ExternalWritable := 'False'} AT Helper_String : Struct
         String_Maximal { ExternalAccessible := 'False'; ExternalVisible := 'False'; ExternalWritable := 'False'} : Byte;
         String_Actual { ExternalAccessible := 'False'; ExternalVisible := 'False'; ExternalWritable := 'False'} : Byte;
         StringValueArray { ExternalAccessible := 'False'; ExternalVisible := 'False'; ExternalWritable := 'False'} : Array[0..15] of Byte;
      END_STRUCT;
   END_VAR
   VAR
      S7ConnTON {OriginalPartName := 'IEC_TIMER'; LibVersion := '1.0'; ExternalAccessible := 'False'; ExternalVisible := 'False'; ExternalWritable := 'False'} : TON_TIME;
   END_VAR

   VAR_TEMP
      i : Int;
      ModBusOK : Bool;
      S7OK : Bool;
   END_VAR


BEGIN
	//Author: Miklos Boros (miklos.boros@esss.se), Copyrigth 2017-2019 by European Spallation Source, Lund
	//This block was generated by PLCFactory
	//Description: This FB checks the EPICS configuration and outputs the result into EPICS_DebuggerResult.

	//DO NOT Modify this block!!!


	#GetChecksum_Instance(Scope:=#scope,
	                      Done=>#done,
	                      Busy=>#busy,
	                      Error=>#error,
	                      Status=>#memErrStatus,
	                      Checksum:="EPICS_DebuggerResult".EPICS_Debugger_Checksum);


	#CheckUtilitiesTON(IN:="Utilities".Square_100ms,
	                   PT:=T#200ms,
	                   Q=>#UtilSquareErrorTON);

	#CheckUtilitiesTON2(IN := NOT "Utilities".Square_100ms,
	                   PT := T#200ms,
	                   Q => #UtilSquareErrorTON2);


	#ModBus_TON(IN := #ModBus_wordsave = "EPICSToPLC"."Word"[2],
	            PT := T#5s);


	IF ("Utilities".AlwaysOn = FALSE) THEN
	    "EPICS_DebuggerResult".#EPICS_Debugger_UtilitiesCall := 'ERROR: FunctionBlock: "_UilitiesFB" is called with a wrong InstanceDB. Call it with the existing iDB named: "Utilities" AND check if the System Memory bits and the System Clock byte is enabled!';
	ELSE
	    IF (#UtilSquareErrorTON OR #UtilSquareErrorTON2) THEN
	        "EPICS_DebuggerResult".#EPICS_Debugger_UtilitiesCall := 'ERROR: FunctionBlock: "_UilitiesFB" is called with a wrong InstanceDB. Call it with the existing iDB named: "Utilities" AND check if the System Memory bits and the System Clock byte is enabled!';
	    ELSE
	        "EPICS_DebuggerResult".#EPICS_Debugger_UtilitiesCall := 'OK: EPICS Utilities works as expected.';

	    END_IF;
	END_IF;

	IF ("Utilities".EPICS_Device_calls_precessed) THEN
	    "EPICS_DebuggerResult".#EPICS_Debugger_DeviceCalls := 'OK: "EPICS_device_calls" is called as expected.';
	ELSE
	    "EPICS_DebuggerResult".#EPICS_Debugger_DeviceCalls := 'ERROR: "EPICS_device_calls" is not called in OB1!';
	END_IF;

	IF (("EPICSToPLC"."Word"[0] = "PLCToEPICS"."Word"[0]) AND ("EPICSToPLC"."Word"[1] = "PLCToEPICS"."Word"[1])) THEN
	    "EPICS_DebuggerResult".#EPICS_Debugger_IOCHash := 'OK: IOC and PLC hash are equal.';
	ELSE
	    "EPICS_DebuggerResult".#EPICS_Debugger_IOCHash := 'ERROR: IOC and PLC hash are NOT equal!';
	END_IF;

	IF (#ModBus_TON.Q) THEN
	    "EPICS_DebuggerResult".#EPICS_Debugger_ModBusHeartBeat := 'ERROR: The IOC is not sending any HeartBeat via ModBus!';
	    #ModBusOK := FALSE;
	ELSE
	    "EPICS_DebuggerResult".#EPICS_Debugger_ModBusHeartBeat := 'OK: ModBus HeartBeat is received as expected.';
	    #ModBusOK := TRUE;
	END_IF;

	#S7ConnTON(IN := NOT "_CommsPLC_EPICS_DB".SendDone, PT := T#3s);

	IF ("_CommsPLC_EPICS_DB".BytesToSend > 0) THEN

	    IF (#S7ConnTON.Q) THEN
	        "EPICS_DebuggerResult".EPICS_Debugger_S7Connection := 'ERROR: EPICS S7 connection can not send Status variables!';
	        #S7OK := FALSE;
	    ELSE
	        "EPICS_DebuggerResult".EPICS_Debugger_S7Connection := 'OK: EPICS S7 works as expected.';
	        #S7OK := TRUE;

	    END_IF;
	ELSE
	    "EPICS_DebuggerResult".EPICS_Debugger_S7Connection := 'OK: EPICS S7 disabled, there is no Status variable to send.';
	    #S7OK := TRUE;
	END_IF;

	IF (#ModBusOK AND #S7OK) THEN
	    "EPICS_DebuggerResult".EPICS_Debugger_EPICS_GeneralState := 'OK. EPICS IOC communication is ONLINE.';
	END_IF;

	IF (#ModBusOK AND NOT #S7OK) THEN
	    "EPICS_DebuggerResult".EPICS_Debugger_EPICS_GeneralState := 'ERROR. ModBus seems to be working but S7 TCP is blocked. Try to check your PLC router IP.';
	END_IF;

	IF (NOT #ModBusOK AND #S7OK) THEN
	    "EPICS_DebuggerResult".EPICS_Debugger_EPICS_GeneralState := 'ERROR. ModBus seems to be offline. Waiting for IOC to finish connecting to the PLC.';
	END_IF;

	IF ( NOT #ModBusOK AND NOT #S7OK) THEN
	    "EPICS_DebuggerResult".EPICS_Debugger_EPICS_GeneralState := 'ERROR. Both ModBus and S7 TCP seems to be offline. Check if your IOC is running and if it is connected to the right PLC interface. Your HardwareID comes from CCDB!';
	END_IF;

	"EPICS_DebuggerResult".EPICS_ModbusPort := "_CommsPLC_EPICS_DB".MBPort;
	"EPICS_DebuggerResult".EPICS_S7Port := "_CommsPLC_EPICS_DB".S7Port;
	"EPICS_DebuggerResult".EPICS_PLC_EthernetInterface :=  "_CommsPLC_EPICS_DB".InterfaceID;


	#ModBus_wordsave := "EPICSToPLC"."Word"[2];


END_FUNCTION_BLOCK
DATA_BLOCK "EPICS_DebuggerFB_iDB"
{ S7_Optimized_Access := 'TRUE' }
VERSION : 0.1
NON_RETAIN
"EPICS_DebuggerFB"

BEGIN

END_DATA_BLOCK
ORGANIZATION_BLOCK "EPICS_DebuggerOB"
TITLE = "Main Program Sweep (Cycle)"
{ S7_Optimized_Access := 'TRUE' }
VERSION : 0.1

BEGIN
	//Author: Miklos Boros (miklos.boros@esss.se), Copyrigth 2017-2019 by European Spallation Source, Lund
	//This block was generated by PLCFactory
	//Description: This OB is a cyclic OB called in every PLC cycle and EPICS_DebuggerFB checks the EPICS configuration.

	//DO NOT Modify this block!!!
	"EPICS_DebuggerFB_iDB"();


END_ORGANIZATION_BLOCK
DATA_BLOCK "EPICSToPLC"
{ S7_Optimized_Access := 'FALSE' }
VERSION : 0.1
//########## EPICS->PLC datablock ##########
   STRUCT
      "Word" { ExternalAccessible := 'False'; ExternalVisible := 'False'; ExternalWritable := 'False'; } : Array[0..27] of Word;
   END_STRUCT;

BEGIN

END_DATA_BLOCK

DATA_BLOCK "PLCToEPICS"
{ S7_Optimized_Access := 'FALSE' }
VERSION : 0.1
NON_RETAIN
//########## PLC->EPICS datablock ##########
   STRUCT
      "Word" { ExternalAccessible := 'False'; ExternalVisible := 'False'; ExternalWritable := 'False'; } : Array[0..89] of Word;
   END_STRUCT;

BEGIN

END_DATA_BLOCK

FUNCTION "_CommsEPICS" : Void
{ S7_Optimized_Access := 'TRUE' }
VERSION : 0.1
   VAR_TEMP
      PLC_Hash : DInt;
   END_VAR

BEGIN
	//Heartbeat PLC->EPICS
	IF "Utilities".Pulse_1s THEN
	    "PLCToEPICS"."Word"[2] := "PLCToEPICS"."Word"[2] + 1;
	    IF "PLCToEPICS"."Word"[2] >= 32000 THEN
	        "PLCToEPICS"."Word"[2] := 0;
	    END_IF;
	END_IF;

	// PLC Factory commit ID: N/A
	// PLC Hash (Generated by PLC Factory)
	#PLC_Hash := DINT#1347332123;

	// Send the PLC Hash to the EPICS IOC
	"PLCToEPICS"."Word"[1] := DINT_TO_WORD(#PLC_Hash);
	"PLCToEPICS"."Word"[0] := DINT_TO_WORD(SHR(IN := #PLC_Hash, N := 16));

	// Call the comms block to provide PLC<->EPICS comms
	"_CommsPLC_EPICS_DB"(Enable         := "Utilities".AlwaysOn,
	                     SendTrigger    := "Utilities".Pulse_200ms,
	                     BytesToSend    := 180,
	                     InterfaceID    := 72,
	                     S7ConnectionID := 256,
	                     MBConnectionID := 255,
	                     S7Port         := 2000,
	                     MBPort         := 502,
	                     PLCToEPICSData := "PLCToEPICS"."Word",
	                     EPICSToPLCData := "EPICSToPLC"."Word");

END_FUNCTION
